// TIA Portal project "Soru2" (V15)

(* hardware
DEVICE "S7-1200 station_1"  S7-1200 Station
   slot 0: "Rack_0"  S7-1200 Rack  Rack  V1.0
   slot 1: "PLC_1"  CPU 1214C DC/DC/DC  6ES7 214-1AG40-0XB0  V4.2
*)

// ===== PLC "PLC_1"  CPU 1214C DC/DC/DC =====

VAR_GLOBAL   // PLC tag table "Default tag table"
   "Alarm" AT %Q0.0 : Bool;
   "Baslat" AT %I0.1 : Bool;
   "Dur" AT %I0.0 : Bool;
END_VAR

// folder: System blocks/Program resources

DATA_BLOCK "zaman"   // DB1
{ S7_Optimized_Access := 'TRUE' }
AUTHOR : Simatic
FAMILY : IEC
NAME : IEC_TMR
VERSION : 1.0
// stored: InstanceOfName IEC_TIMER
"IEC_TIMER"
BEGIN
END_DATA_BLOCK

// folder: (top level)

ORGANIZATION_BLOCK "Main"   // OB1, LAD, ProgramCycle
TITLE = "Main Program Sweep (Cycle)"
{ S7_Optimized_Access := 'TRUE' }
VERSION : 0.1
   VAR_INPUT
      Initial_Call : Bool;   // Initial call of this OB
      Remanence : Bool;   // =True, if remanent data are available
   END_VAR
BEGIN

REGION Network 1: Zamna Rölesi ayarlamsı
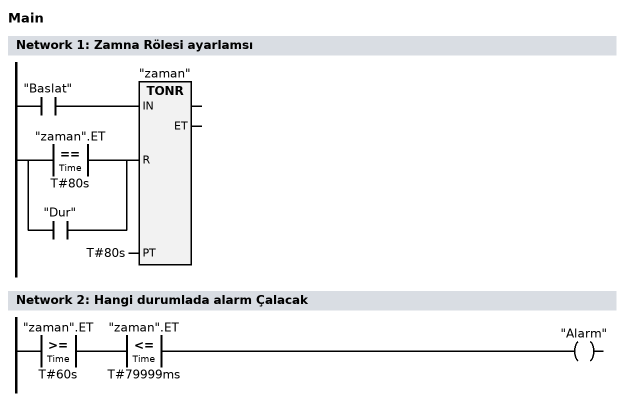
   "zaman".TONR(IN := "Baslat", R := ("zaman".ET = T#80s) OR "Dur", PT := T#80s);
END_REGION

REGION Network 2: Hangi durumlada alarm Çalacak
   RUNG wire#powerrail
      { S7_Templates := "SrcType := Time" } GE_Contact(in1 := "zaman".ET, in2 := T#60s)
      { S7_Templates := "SrcType := Time" } LE_Contact(in1 := "zaman".ET, in2 := T#79999ms)
      Coil( "Alarm" )
   END_RUNG
   // the same network as SCL:
   "Alarm" := ("zaman".ET >= T#60s) AND ("zaman".ET <= T#79999ms);
END_REGION
END_ORGANIZATION_BLOCK